Staubli VAL3: home.dtx

num nKey = 271
public num nPage = 10
num nRefresh = 33.117
num nTime = 1
num nValue[4]
  [0] = 1
  [1] = 2
  [2] = 3
  [3] = 4
public string sItems
string sMenu
string sMessage
string sVersion = "valClean 7.3.1.8"
string sMenu8[8]
string sSession
string sPathSession
string sDeeperSession
bool bButton[8]
  [0] = true
  [1] = true
  [2] = true
  [4] = true
  [5] = true
  [6] = true
  [7] = true
